(* IEC 61131-3 sources: Industry-PLC-LLM/data/PLCBEAD_repo/PLCBEAD_PLCEmbed-main/PLC-BEAD/Source/GEB/ISC_HEX, 1 file *)

(* ---- ISC_HEX.ST ---- *)
FUNCTION ISC_HEX:BOOL

	VAR_INPUT
		IN :	BYTE;
	END_VAR

	ISC_HEX := (IN > BYTE#47 AND IN < BYTE#58) OR (IN > BYTE#64 AND IN < BYTE#71) OR (IN > BYTE#96 AND IN < BYTE#103);

END_FUNCTION

PROGRAM program0
	VAR
		IN : BYTE;
		OUT : BOOL;
	END_VAR

	OUT := ISC_HEX(IN);
END_PROGRAM
